// TwinCAT 3 PLC project PLC_01
// ProgramVersion: 3.1.4023.0
// libraries:
//   Tc2_Standard, * (Beckhoff Automation GmbH)
//   Tc2_System, * (Beckhoff Automation GmbH)
//   Tc3_Module, * (Beckhoff Automation GmbH)
// project tree:
//   / PlcTask.TcTTO
//   POUs/ MAIN.TcPOU
// real-time tasks:
//   TASK PlcTask: cycle T#10ms, priority 20, ADS port 350

CONFIGURATION PLC_01
    RESOURCE PLC ON TwinCAT3
        TASK PlcTask(INTERVAL := T#10ms, PRIORITY := 20);
        PROGRAM MAIN WITH PlcTask : MAIN;
    END_RESOURCE
END_CONFIGURATION

// ---- POUs/MAIN.TcPOU
PROGRAM MAIN
VAR
	
FB_TON_01 : TON ;  															// DECLARAÇÃO TON 01 


Botao_In        : BOOL ;													//	Inicio do Tempo 	
Botao_Out       : BOOL ; 													//	Saída Ativa quando o tempo for alcançado 	
T_Presete_Time  : TIME := T#120S ;											//	Valoe que o bloco deve alcançar 
T_Elapse_Time   : TIME ; 													//	Tempo decorrido desde a ativação 
	
	
END_VAR

FB_TON_01 (IN:= Botao_In, PT:= T_Presete_Time, Q=> Botao_Out, ET => T_Elapse_Time);

END_PROGRAM
